SUBAPPLICATION Uebung_020f4_AX (* DigitalInput_I1 auf DataPanel_1A; BLINKER *)
  (* Standard: 61499-2; Description: Copyright (c) 2023 Meisterschulen am Ostbahnhof This program and the accompanying materials are made available under the terms of the Eclipse Public License 2.0 which is available at https://www.eclipse.org/legal/epl-2.0/ SPDX-License-Identifier: EPL-2.0 *)
  (* Version 1.0, 2023-10-23, Franz Höpfinger, Meisterschulen am Ostbahnhof, initial API and implementation and/or initial documentation *)
  PACKAGE Uebungen;
  IMPORT DataPanel::io::MI::DQ::DataPanel_MI_DO::DigitalOutput_1A;
  IMPORT DataPanel::io::MI::const::MI::MI_00;
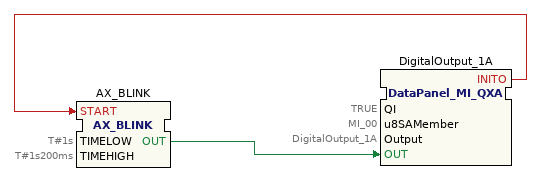
  FBS
    AX_BLINK : adapter::events::unidirectional::signals::AX_BLINK(TIMELOW := T#1s, TIMEHIGH := T#1s200ms);
    DigitalOutput_1A : DataPanel::io::MI::DQ::DataPanel_MI_QXA(QI := TRUE, u8SAMember := MI_00, Output := DigitalOutput_1A);
  END_FBS
  EVENT_CONNECTIONS
    DigitalOutput_1A.INITO TO AX_BLINK.START;
  END_CONNECTIONS
  ADAPTER_CONNECTIONS
    AX_BLINK.OUT TO DigitalOutput_1A.OUT;
  END_CONNECTIONS
END_SUBAPPLICATION
